INTERFACE I_Drive

{attribute 'monitoring':='call'}
PROPERTY Active : BOOL
GET
END_GET
END_PROPERTY

{attribute 'monitoring':='call'}
PROPERTY Error : BOOL
GET
END_GET
END_PROPERTY

METHOD reset : BOOL
VAR_INPUT
END_VAR
END_METHOD

METHOD ABSTRACT stop : BOOL
VAR_INPUT
END_VAR
END_METHOD

END_INTERFACE

(* stored: Version 1.1.0.1, ProductVersion 3.1.4024.11
   Itf I_Drive: Id {2c083758-60a9-42e5-a9a1-167bf3458c3a}
   Property Active: Id {e3ee71e9-61f6-4f82-8a9c-581168957511}
   Get Get: Id {4055766e-8def-4c11-a4aa-41a5f78c487a}
   Property Error: Id {44982ee4-6b3b-43ac-b3a6-0ca396eb993d}
   Get Get: Id {c76cc53d-1c48-418b-a9be-3cb0b16d9e08}
   Method reset: Id {bcb8f5dc-bcb0-4e14-825d-9286830c3b35}
   Method stop: Id {71ff8128-8f23-47f2-97f3-4bd7159ef989} *)
